FUNCTION F_ResetExternalSubsystemError : BOOL
(**************************************************************************************
 * 	Application		:	BoxControl Framework
 *	Revision		:	$Revision: 404529 $
 *	Revision date	:	$Date: 2018-04-23 08:21:38 +0200 (Mo., 23 Apr 2018) $
 *	Last changed by	:	$Author: b7bolm $
 *	URL				:	$URL: http://almscdc.swisslog.com/repo/SWPD/Development/BoxControlFramework/20_Release/trunk/01_Software/BCF/BCF/JumpStart/20_Product/10_App/15_Subsystem/10_Lib/10_Conv/10_Functions/F_ResetExternalSubsystemError.TcPOU $
 *
 *	Purpose			:	Reset external error
 *						Add an External error, which will be reported over the configured
 *						position.
 *						
 *
 * ------------------------------------------------------------------------------------
 *	Copyright Swisslog [IP AG], Switzerland. All rights reserved.
 * 
 * ------------------------------------------------------------------------------------
 *	
 * 	Revision History: 
 *
 * 	VERSION			DATE			INITIALS			DESCRIPTION
 *	0.1				01.01.2001		swl					Example
 *
 **************************************************************************************)
VAR_INPUT
	Reset			: BOOL;
END_VAR


IF __ISVALIDREF(SubsystemRegistry.rSubsystem) THEN
	// Reset external error on instance
	SubsystemRegistry.rSubsystem.M_ResetExternalError(
		mReset := Reset);
END_IF

END_FUNCTION

(* stored: Version 1.1.0.1, ProductVersion 3.1.4022.12
   POU F_ResetExternalSubsystemError: Id {4f1bc672-12af-4f76-bcb0-dbebc5734ee6}, SpecialFunc None *)
